(* Schneider Machine Expert - Basic project TransportRouteControl, file version 2.9.0.0 *)
(* ProjectInformations: Name=New project *)

HARDWARE
  Cpu 0: TM221CE16R
  EthernetConfiguration: NetworkName=M221, IpAllocationMode=FixedAddress, IpAddress=192.168.50.50, SubnetMask=255.255.255.0
  SerialLineConfiguration: Baud=Baud19200, Parity=ParityEven, DataBits=DataBits8, StopBits=StopBits1, PhysicalMedium=PhysicalMediumRs485, SlaveId=1, Addressing=SlaveAddressing
  MastTask: UsePeriodScanMode=true, PeriodScan=10
  FastTask: Period=255
  CpuBehavior: StartingMode=StartAsPreviousState, AutoSaveRamOnEeprom=true, WatchdogPeriod=250

SYMBOLS  (address, symbol, comment, settings)
  %M0       PART_AVAILABLE
  %M1       CONTROLLER_ACTIVE
  %MW0      WORK_PIECE_COUNTER
  %MW1      STATE
  %KW0      MODBUS_WRITE_VALUE  [Value=2]
  %TM0      TRANSPORTTIMER  "Timer for Rotating the Belt."  [Preset=3000, Base=OneMilliSeconds]
  %TRANSPORTROUTECONTROL0 TRANSPORT_ROUTE_CONTROLLER  [UserDefineFunctionPouName=TRANSPORTROUTECONTROL]
  %I0.0     SLIDER_LIMIT_SWITCH
  %I0.1     BELT_LIGHT_BARRIER
  %I0.2     PALLET_LIGHT_BARRIER_TOP
  %I0.3     PALLET_LIGHT_BARRIER_BOTTOM
  %Q0.0     MOTOR_SLIDER_PUSHER
  %Q0.1     MOTOR_BELT
  %Q0.2     VALVE_SEPARATOR
  %IWN300.0.1   [Channel=READ_VALUE]
  %QWN300.1.0   [Channel=WRITE_VALUE]

POU main
  (* SectionNumber=1 *)

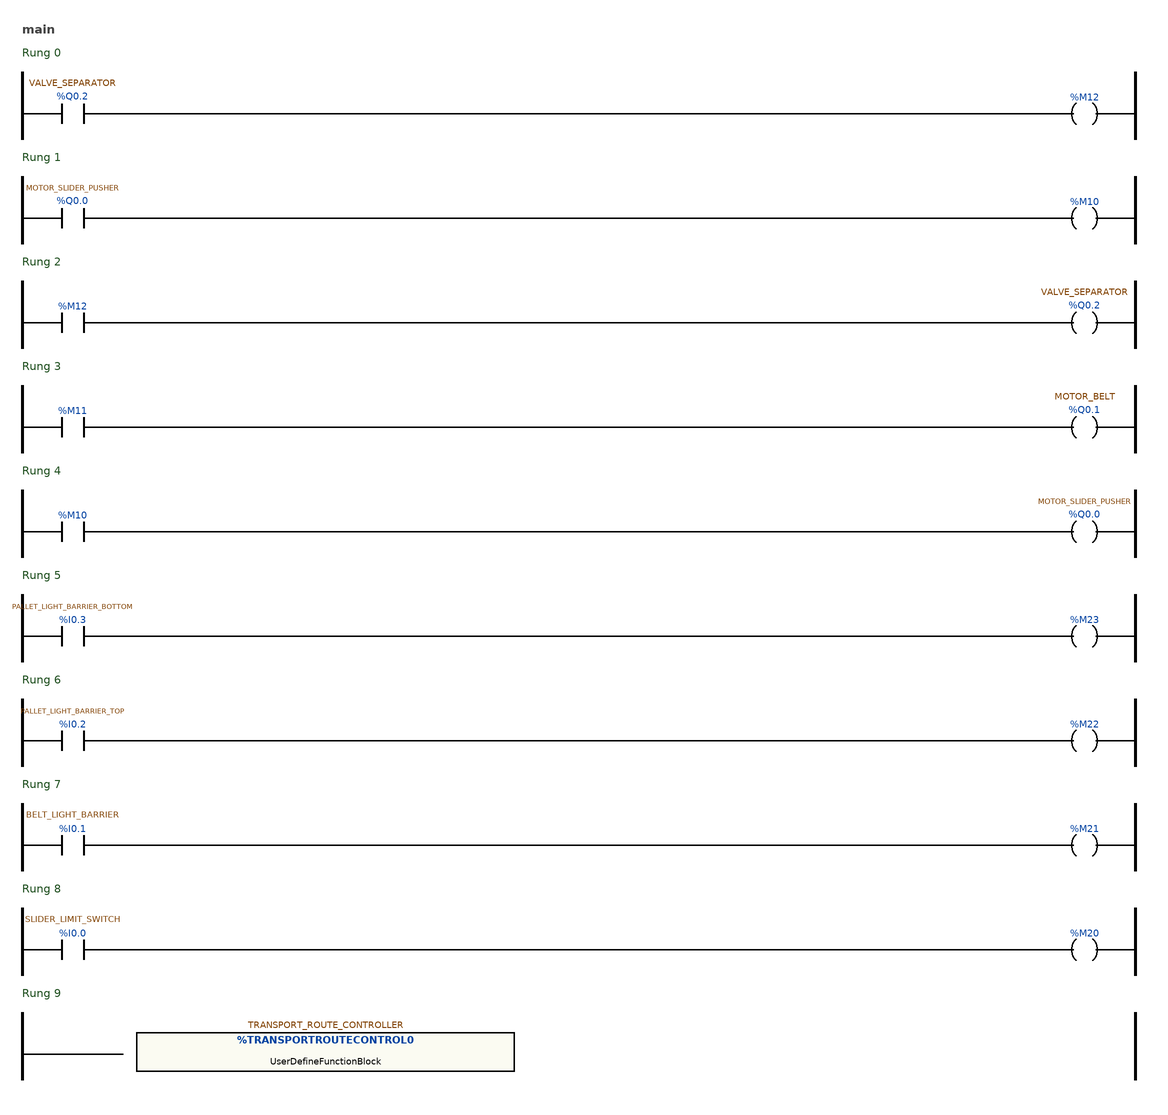

// Rung 0
  LD %Q0.2                (* VALVE_SEPARATOR *)
  ST %M12
  // as ST:
  //   %M12 := VALVE_SEPARATOR;

// Rung 1
  LD %Q0.0                (* MOTOR_SLIDER_PUSHER *)
  ST %M10
  // as ST:
  //   %M10 := MOTOR_SLIDER_PUSHER;

// Rung 2
  LD %M12
  ST %Q0.2                (* VALVE_SEPARATOR *)
  // as ST:
  //   VALVE_SEPARATOR := %M12;

// Rung 3
  LD %M11
  ST %Q0.1                (* MOTOR_BELT *)
  // as ST:
  //   MOTOR_BELT := %M11;

// Rung 4
  LD %M10
  ST %Q0.0                (* MOTOR_SLIDER_PUSHER *)
  // as ST:
  //   MOTOR_SLIDER_PUSHER := %M10;

// Rung 5
  LD %I0.3                (* PALLET_LIGHT_BARRIER_BOTTOM *)
  ST %M23
  // as ST:
  //   %M23 := PALLET_LIGHT_BARRIER_BOTTOM;

// Rung 6
  LD %I0.2                (* PALLET_LIGHT_BARRIER_TOP *)
  ST %M22
  // as ST:
  //   %M22 := PALLET_LIGHT_BARRIER_TOP;

// Rung 7
  LD %I0.1                (* BELT_LIGHT_BARRIER *)
  ST %M21
  // as ST:
  //   %M21 := BELT_LIGHT_BARRIER;

// Rung 8
  LD %I0.0                (* SLIDER_LIMIT_SWITCH *)
  ST %M20
  // as ST:
  //   %M20 := SLIDER_LIMIT_SWITCH;

// Rung 9
  LD 1
  BLK_UDFB 3
  LD 1
  ST %UDF1.PARAMW0:X0
  LD 1
  ST %UDF1.PARAMW0:X8
  [ %UDF1.RETW0 := %UDF2.RETW0 ]
  [ %UDF1.RETW1 := %UDF2.RETW1 ]
  [ %UDF1.RETW2 := %UDF2.RETW2 ]
  [ %UDF1.RETW3 := %UDF2.RETW3 ]
  UDF1
  [ %UDF2.RETW0 := %UDF1.RETW0 ]
  [ %UDF2.RETW1 := %UDF1.RETW1 ]
  [ %UDF2.RETW2 := %UDF1.RETW2 ]
  [ %UDF2.RETW3 := %UDF1.RETW3 ]
  END_BLK_UDFB 3

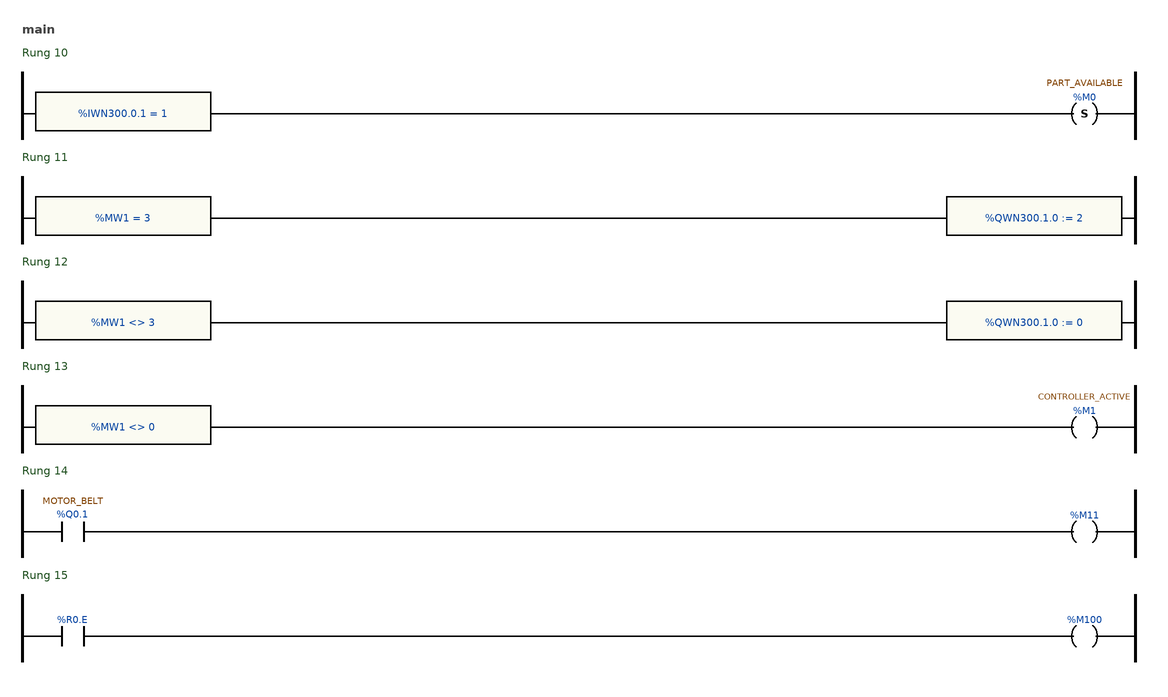

// Rung 10
  LD [ %IWN300.0.1 = 1 ]
  S %M0                   (* PART_AVAILABLE *)
  // as ST:
  //   IF %IWN300.0.1 = 1 THEN PART_AVAILABLE := TRUE; END_IF;

// Rung 11
  LD [ %MW1 = 3 ]         (* STATE *)
  [ %QWN300.1.0 := 2 ]
  // as ST:
  //   IF STATE = 3 THEN %QWN300.1.0 := 2; END_IF;

// Rung 12
  LD [ %MW1 <> 3 ]        (* STATE *)
  [ %QWN300.1.0 := 0 ]
  // as ST:
  //   IF STATE <> 3 THEN %QWN300.1.0 := 0; END_IF;

// Rung 13
  LD [ %MW1 <> 0 ]        (* STATE *)
  ST %M1                  (* CONTROLLER_ACTIVE *)
  // as ST:
  //   CONTROLLER_ACTIVE := STATE <> 0;

// Rung 14
  LD %Q0.1                (* MOTOR_BELT *)
  ST %M11
  // as ST:
  //   %M11 := MOTOR_BELT;

// Rung 15
  LD %R0.E
  ST %M100
  // as ST:
  //   %M100 := %R0.E;

UserFunctionBlockPou TRANSPORTROUTECONTROL
  (* SectionNumber=3 *)

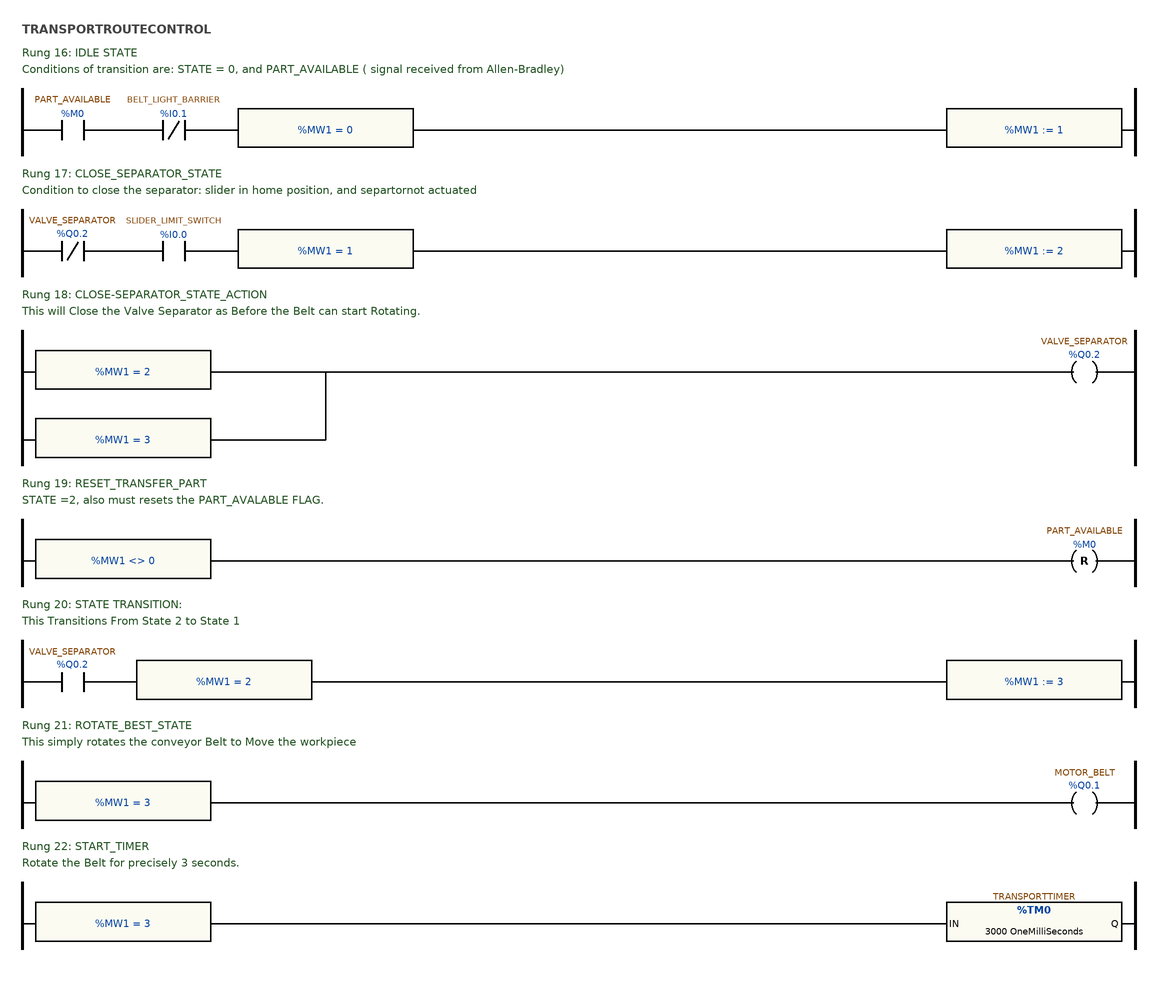

// Rung 16: IDLE STATE
// Conditions of transition are: STATE = 0, and PART_AVAILABLE ( signal received from Allen-Bradley)
  LD %M0                  (* PART_AVAILABLE *)
  ANDN %I0.1              (* BELT_LIGHT_BARRIER *)
  AND [ %MW1 = 0 ]        (* STATE *)
  [ %MW1 := 1 ]           (* STATE *)
  // as ST:
  //   IF PART_AVAILABLE AND NOT BELT_LIGHT_BARRIER AND STATE = 0 THEN STATE := 1; END_IF;

// Rung 17: CLOSE_SEPARATOR_STATE
// Condition to close the separator: slider in home position, and separtornot actuated
  LDN %Q0.2               (* VALVE_SEPARATOR *)
  AND %I0.0               (* SLIDER_LIMIT_SWITCH *)
  AND [ %MW1 = 1 ]        (* STATE *)
  [ %MW1 := 2 ]           (* STATE *)
  // as ST:
  //   IF NOT VALVE_SEPARATOR AND SLIDER_LIMIT_SWITCH AND STATE = 1 THEN STATE := 2; END_IF;

// Rung 18: CLOSE-SEPARATOR_STATE_ACTION
// This will Close the Valve Separator as Before the Belt can start Rotating.
  LD [ %MW1 = 2 ]         (* STATE *)
  OR [ %MW1 = 3 ]         (* STATE *)
  ST %Q0.2                (* VALVE_SEPARATOR *)
  // as ST:
  //   VALVE_SEPARATOR := STATE = 2 OR STATE = 3;

// Rung 19: RESET_TRANSFER_PART
// STATE =2, also must resets the PART_AVALABLE FLAG.
  LD [ %MW1 <> 0 ]        (* STATE *)
  R %M0                   (* PART_AVAILABLE *)
  // as ST:
  //   IF STATE <> 0 THEN PART_AVAILABLE := FALSE; END_IF;

// Rung 20: STATE TRANSITION:
// This Transitions From State 2 to State 1
  LD %Q0.2                (* VALVE_SEPARATOR *)
  AND [ %MW1 = 2 ]        (* STATE *)
  [ %MW1 := 3 ]           (* STATE *)
  // as ST:
  //   IF VALVE_SEPARATOR AND STATE = 2 THEN STATE := 3; END_IF;

// Rung 21: ROTATE_BEST_STATE
// This simply rotates the conveyor Belt to Move the workpiece
  LD [ %MW1 = 3 ]         (* STATE *)
  ST %Q0.1                (* MOTOR_BELT *)
  // as ST:
  //   MOTOR_BELT := STATE = 3;

// Rung 22: START_TIMER
// Rotate the Belt for precisely 3 seconds.
  BLK %TM0                (* TRANSPORTTIMER *)
  LD [ %MW1 = 3 ]         (* STATE *)
  IN
  END_BLK
  // as ST:
  //   TRANSPORTTIMER(IN := STATE = 3);

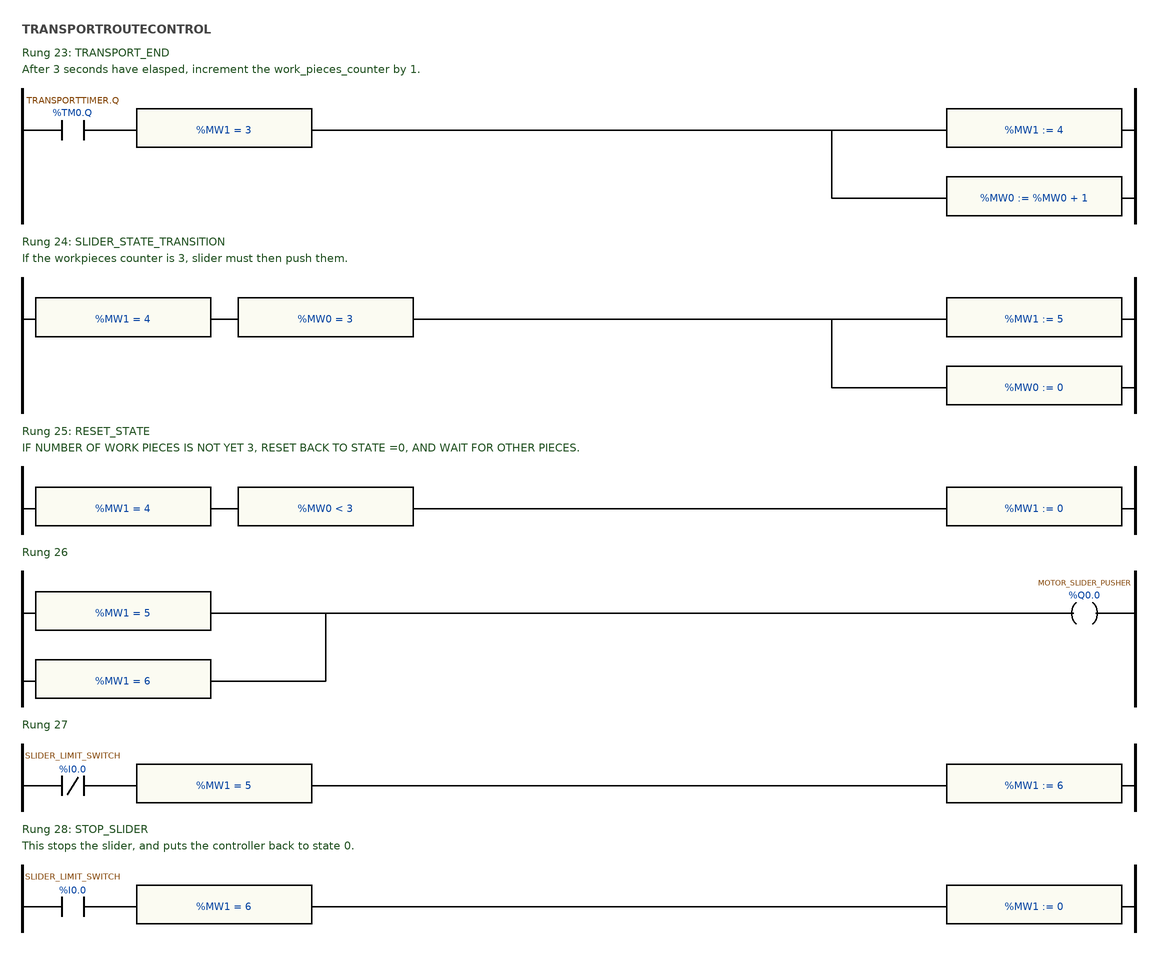

// Rung 23: TRANSPORT_END
// After 3 seconds have elasped, increment the work_pieces_counter by 1.
  LD %TM0.Q               (* TRANSPORTTIMER *)
  AND [ %MW1 = 3 ]        (* STATE *)
  [ %MW1 := 4 ]           (* STATE *)
  [ %MW0 := %MW0 + 1 ]    (* WORK_PIECE_COUNTER, WORK_PIECE_COUNTER *)
  // as ST:
  //   _t1 := TRANSPORTTIMER.Q AND STATE = 3;
  //   IF _t1 THEN STATE := 4; END_IF;
  //   IF _t1 THEN WORK_PIECE_COUNTER := WORK_PIECE_COUNTER + 1; END_IF;

// Rung 24: SLIDER_STATE_TRANSITION
// If the workpieces counter is 3, slider must then push them.
  LD [ %MW1 = 4 ]         (* STATE *)
  AND [ %MW0 = 3 ]        (* WORK_PIECE_COUNTER *)
  [ %MW1 := 5 ]           (* STATE *)
  [ %MW0 := 0 ]           (* WORK_PIECE_COUNTER *)
  // as ST:
  //   _t1 := STATE = 4 AND WORK_PIECE_COUNTER = 3;
  //   IF _t1 THEN STATE := 5; END_IF;
  //   IF _t1 THEN WORK_PIECE_COUNTER := 0; END_IF;

// Rung 25: RESET_STATE
// IF NUMBER OF WORK PIECES IS NOT YET 3, RESET BACK TO STATE =0, AND WAIT FOR OTHER PIECES.
  LD [ %MW1 = 4 ]         (* STATE *)
  AND [ %MW0 < 3 ]        (* WORK_PIECE_COUNTER *)
  [ %MW1 := 0 ]           (* STATE *)
  // as ST:
  //   IF STATE = 4 AND WORK_PIECE_COUNTER < 3 THEN STATE := 0; END_IF;

// Rung 26
  LD [ %MW1 = 5 ]         (* STATE *)
  OR [ %MW1 = 6 ]         (* STATE *)
  ST %Q0.0                (* MOTOR_SLIDER_PUSHER *)
  // as ST:
  //   MOTOR_SLIDER_PUSHER := STATE = 5 OR STATE = 6;

// Rung 27
  LDN %I0.0               (* SLIDER_LIMIT_SWITCH *)
  AND [ %MW1 = 5 ]        (* STATE *)
  [ %MW1 := 6 ]           (* STATE *)
  // as ST:
  //   IF NOT SLIDER_LIMIT_SWITCH AND STATE = 5 THEN STATE := 6; END_IF;

// Rung 28: STOP_SLIDER
// This stops the slider, and puts the controller back to state 0.
  LD %I0.0                (* SLIDER_LIMIT_SWITCH *)
  AND [ %MW1 = 6 ]        (* STATE *)
  [ %MW1 := 0 ]           (* STATE *)
  // as ST:
  //   IF SLIDER_LIMIT_SWITCH AND STATE = 6 THEN STATE := 0; END_IF;
